# EPICS autosave request: stdApp/Db/autoShutter_settings.req
# FILE... autoShutter_settings.req
$(P)$(S)Shtr:Enable
$(P)$(S)Shtr:ThresholdCurrent
file scalcout_settings.req P=$(P)$(S)Shtr:UserArm
file calcout_settings.req P=$(P)$(S)Shtr:EnableOff
